// TIA Portal project "S7netTiaProject(RobotControl)" (V16)

(* hardware
DEVICE "S7-1200 station_1"  S7-1200 Station
   slot 0: "Rack_0"  S7-1200 Rack  Rack  V1.0
   slot 1: "PLC_1"  CPU 1214C DC/DC/DC  6ES7 214-1AG40-0XB0  V4.4
*)

// ===== PLC "PLC_1"  CPU 1214C DC/DC/DC =====

VAR_GLOBAL   // PLC tag table "Default tag table"
   "Tag_1" AT %Q0.0 : Bool;
   "M1" AT %M0.1 : Bool;
   "sum" AT %MW20 : Int;
   "start" AT %M0.0 : Bool;
END_VAR

DATA_BLOCK "DataBlock1"   // DB1
{ S7_Optimized_Access := 'FALSE' }
VERSION : 0.1
   VAR
      Btn1 : Bool := false;
      Btn2 : Bool;
      Btn3 : Bool;
      SQ1 : Bool;
      SQ2 : Bool;
      "Robot proceed" : Bool;
      "Create red" : Bool;
      "Create green" : Bool;
      "Create blue" : Bool;
      "Locate red" : Bool;
      "Locate green" : Bool;
      "Locate blue" : Bool;
      "Conveyor fast" : Bool;
      "Conveyor slow" : Bool;
   END_VAR
BEGIN
END_DATA_BLOCK

ORGANIZATION_BLOCK "Main"   // OB1, LAD, ProgramCycle
TITLE = "Main Program Sweep (Cycle)"
{ S7_Optimized_Access := 'TRUE' }
VERSION : 0.1
   VAR_INPUT
      Initial_Call : Bool;   // Initial call of this OB
      Remanence : Bool;   // =True, if remanent data are available
   END_VAR
BEGIN

REGION Network 1
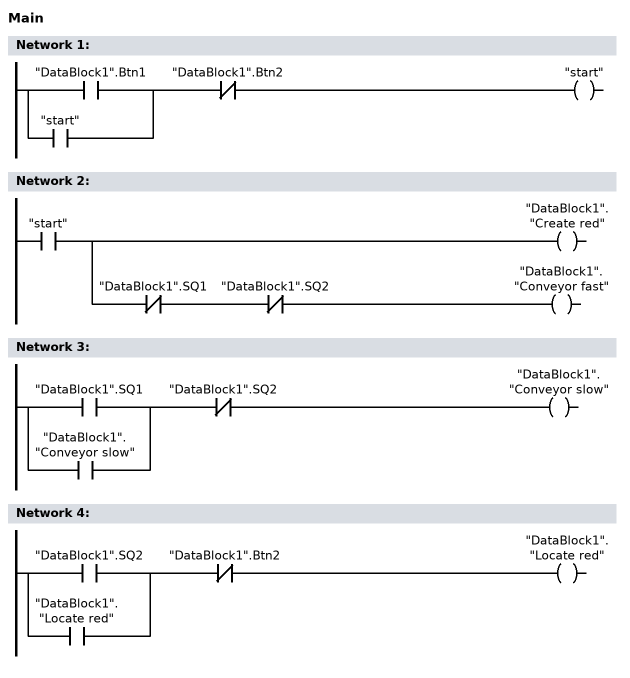
   RUNG wire#powerrail
      Contact( "DataBlock1".Btn1 )
      wire#w1
      I_Contact( "DataBlock1".Btn2 )
      Coil( "start" )
   END_RUNG
   RUNG wire#powerrail
      Contact( "start" )
   END_RUNG wire#w1
   // the same network as SCL:
   "start" := ("DataBlock1".Btn1 OR "start") AND NOT "DataBlock1".Btn2;
END_REGION

REGION Network 2
   RUNG wire#powerrail
      Contact( "start" )
      wire#w1
      Coil( "DataBlock1"."Create red" )
   END_RUNG
   RUNG wire#w1
      I_Contact( "DataBlock1".SQ1 )
      I_Contact( "DataBlock1".SQ2 )
      Coil( "DataBlock1"."Conveyor fast" )
   END_RUNG
   // the same network as SCL:
   "DataBlock1"."Create red" := "start";
   "DataBlock1"."Conveyor fast" := "start" AND NOT "DataBlock1".SQ1 AND NOT "DataBlock1".SQ2;
END_REGION

REGION Network 3
   RUNG wire#powerrail
      Contact( "DataBlock1".SQ1 )
      wire#w1
      I_Contact( "DataBlock1".SQ2 )
      Coil( "DataBlock1"."Conveyor slow" )
   END_RUNG
   RUNG wire#powerrail
      Contact( "DataBlock1"."Conveyor slow" )
   END_RUNG wire#w1
   // the same network as SCL:
   "DataBlock1"."Conveyor slow" := ("DataBlock1".SQ1 OR "DataBlock1"."Conveyor slow") AND NOT "DataBlock1".SQ2;
END_REGION

REGION Network 4
   RUNG wire#powerrail
      Contact( "DataBlock1".SQ2 )
      wire#w1
      I_Contact( "DataBlock1".Btn2 )
      Coil( "DataBlock1"."Locate red" )
   END_RUNG
   RUNG wire#powerrail
      Contact( "DataBlock1"."Locate red" )
   END_RUNG wire#w1
   // the same network as SCL:
   "DataBlock1"."Locate red" := ("DataBlock1".SQ2 OR "DataBlock1"."Locate red") AND NOT "DataBlock1".Btn2;
END_REGION
END_ORGANIZATION_BLOCK